FUNCTION_BLOCK MECH2_DIAG (* Diagnostics for a Bidirectional Mechanism (Clocked) *)
  (* Standard: 61499-1; Classification: Diagnostics; ApplicationDomain: Mechanisms *)
  (* Version 0.1, 2004-10-20, JHC, Rockwell Automation, Renamed to replace old MECH2_DIAG. *)
  (* Version 0.0, 2004-08-26, JHC, Rockwell Automation, Derived from MECH2_DIAG. *)
  (* Compiler header: package fb.rt.mva; import fb.rt.math.*; *)
  (* Compiler Java Sun JDK 1.4.2 *)
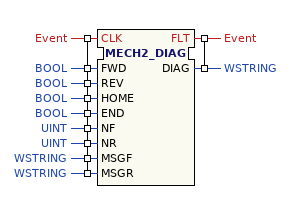
  EVENT_INPUT
    CLK WITH HOME, END, NR, FWD, REV, NF, MSGF, MSGR; (* Diagnostic Clock *)
  END_EVENT
  EVENT_OUTPUT
    FLT WITH DIAG; (* Fault Indication *)
  END_EVENT
  VAR_INPUT
    FWD : BOOL; (* Forward Actuation Command from Controller *)
    REV : BOOL; (* Reverse Actuation Command from Controller *)
    HOME : BOOL; (* HOME(Fully Retracted)Sensor *)
    END : BOOL; (* END(Fully Advanced)Sensor *)
    NF : UINT; (* Forward Motion Timeout Period in CLK cycles *)
    NR : UINT; (* Reverse Motion Timeout Period in CLK cycles *)
    MSGF : WSTRING := "TIMEOUT_ADVANCING"; (* Message for fault on forward motion *)
    MSGR : WSTRING := "TIMEOUT_RETRACTING"; (* Message for fault on reverse motion *)
  END_VAR
  VAR_OUTPUT
    DIAG : WSTRING; (* Diagnostic String *)
  END_VAR
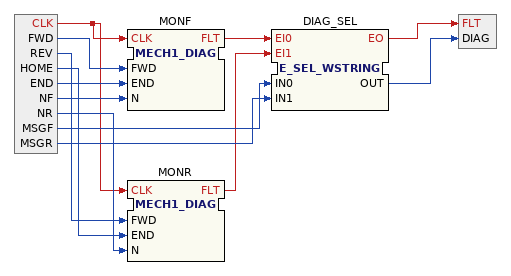
  FBS
    MONF : MECH1_DIAG; (* Monitor Forward Motion *)
    MONR : MECH1_DIAG; (* Monitor reverse motion *)
    DIAG_SEL : E_SEL_WSTRING; (* Diagnostic String Selector *)
  END_FBS
  EVENT_CONNECTIONS
    MONF.FLT TO DIAG_SEL.EI0;
    MONR.FLT TO DIAG_SEL.EI1;
    DIAG_SEL.EO TO FLT;
    CLK TO MONF.CLK;
    CLK TO MONR.CLK;
  END_CONNECTIONS
  DATA_CONNECTIONS
    FWD TO MONF.FWD;
    END TO MONF.END;
    REV TO MONR.FWD;
    HOME TO MONR.END;
    MSGF TO DIAG_SEL.IN0;
    MSGR TO DIAG_SEL.IN1;
    DIAG_SEL.OUT TO DIAG;
    NF TO MONF.N;
    NR TO MONR.N;
  END_CONNECTIONS
END_FUNCTION_BLOCK
